TYPE T_CRYO_CRYOTELGT_CMD :
STRUCT
	cmd:		STRING	:= '';	// Command to send
	nReplies:	INT	:= 1;	// # of Replies
END_STRUCT
END_TYPE

(* stored: Version 1.1.0.1, ProductVersion 3.1.4024.12
   DUT T_CRYO_CRYOTELGT_CMD: Id {b687f34e-eaa3-4f0d-a269-16b9339bccd1} *)
